// TIA Portal V20 export
DATA_BLOCK "SBK9"   // DB293
// stored: MemoryReserve 100
   VAR
      "X1-1 SAFETY DOOR LOCK1.INPUT" : Bool;
      "X2-1 SAFETY DOOR LOCK2.INPUT" : Bool;
      "X3-1 SAFETY DOOR LOCK3.INPUT" : Bool;
      "X4-1 SPARE" : Bool;
      "X1-2 SAFETY DOOR LOCK1.INPUT" : Bool;
      "X2-2 SAFETY DOOR LOCK2.INPUT" : Bool;
      "X3-2 SAFETY DOOR LOCK3.INPUT" : Bool;
      "X4-2 SPARE" : Bool;
   END_VAR
BEGIN
END_DATA_BLOCK
